// TIA Portal V19 export
TYPE "Tel393Out_PM"
// stored: Access Published
   STRUCT
      CU_STW1 : Struct   // Control word 1, Control Unit
         reserved_Bit08 : Bool;   // Reserved
         reserved_Bit09 : Bool;   // Reserved
         ackAutoSuppressed : Bool;   // Acknowledgment automatically suppressed
         reserved_Bit11 : Bool;   // Reserved
         masterSignOfLifeBit0 : Bool;   // Master sign-of-life bit 0
         masterSignOfLifeBit1 : Bool;   // Master sign-of-life bit 1
         masterSignOfLifeBit2 : Bool;   // Master sign-of-life bit 2
         masterSignOfLifeBit3 : Bool;   // Master sign-of-life bit 3
         syncFlag : Bool;   // This signal is used to synchonize the joint system time between the controller and drive unit BI: p 0681[0]
         rtcPing : Bool;   // This signal is used to set the UTC time using the Ping event BI: p 3104
         esrTrigger : Bool;   // ESR-Trigger
         reserved_Bit03 : Bool;   // Reserved
         reserved_Bit04 : Bool;   // Reserved
         reserved_Bit05 : Bool;   // Reserved
         reserved_Bit06 : Bool;   // Reserved
         acknowledge : Bool;   // 0 --> 1 = Acknowledge faults (Acknowledge fault. If the ON command is still active, the inverter switches to "closing lockout" state) p 2103[0] = r 2090.7
      END_STRUCT;
      A_DIGITAL : Struct   // Digital output (16-bit)
         reserved_Bit08 : Bool;   // Reserved
         reserved_Bit09 : Bool;   // Reserved
         reserved_Bit10 : Bool;   // Reserved
         reserved_Bit11 : Bool;   // Reserved
         reserved_Bit12 : Bool;   // Reserved
         reserved_Bit13 : Bool;   // Reserved
         reserved_Bit14 : Bool;   // Reserved
         reserved_Bit15 : Bool;   // Reserved
         digitalOutput8 : Bool;   // Digital output 8 (DI/DO 8); p0738 = r2091.0
         digitalOutput9 : Bool;   // Digital output 9 (DI/DO 9); p0739 = r2091.1
         digitalOutput10 : Bool;   // Digital output 10 (DI/DO 10); p0740 = r2091.2
         digitalOutput11 : Bool;   // Digital output 11 (DI/DO 11); p0741 = r2091.3
         digitalOutput12 : Bool;   // Digital output 12 (DI/DO 12); p0742 = r2091.4
         digitalOutput13 : Bool;   // Digital output 13 (DI/DO 13); p0743 = r2091.5
         digitalOutput14 : Bool;   // Digital output 14 (DI/DO 14); p0744 = r2091.6
         digitalOutput15 : Bool;   // Digital output 15 (DI/DO 15); p0745 = r2091.7
      END_STRUCT;
      A_DIGITAL_1 : Struct   // Digital output (16-bit)
         digitalOutput16 : Bool;   // Digital output 16 (DI/DO 16); p0746 = r2092.8
         reserved_Bit09 : Bool;   // Reserved
         reserved_Bit10 : Bool;   // Reserved
         reserved_Bit11 : Bool;   // Reserved
         reserved_Bit12 : Bool;   // Reserved
         reserved_Bit13 : Bool;   // Reserved
         reserved_Bit14 : Bool;   // Reserved
         reserved_Bit15 : Bool;   // Reserved
         "2ndacknowledge" : Bool;   // Set p2104 with r2092.0
         PathTestAxis1 : Bool;   // Set the Axis Stop test with r2092.1 from CU
         PathTestAxis2 : Bool;   // Set the Axis Stop test with r2092.2 from CU
         PathTestAxis3 : Bool;   // Set the Axis Stop test with r2092.3 from CU
         PathTestAxis4 : Bool;   // Set the Axis Stop test with r2092.4 from CU
         reserved_Bit05 : Bool;   // Reserved
         reserved_Bit06 : Bool;   // Reserved
         reserved_Bit07 : Bool;   // Reserved
      END_STRUCT;
      MT_STW : Struct   // Measuring probe control word
         risProbe1 : Bool;   // Activation of measuring time determination with the next rising edge
         risProbe2 : Bool;   // Activation of measuring time determination with the next rising edge
         risProbe3 : Bool;   // Activation of measuring time determination with the next rising edge
         risProbe4 : Bool;   // Activation of measuring time determination with the next rising edge
         risProbe5 : Bool;   // Activation of measuring time determination with the next rising edge
         risProbe6 : Bool;   // Activation of measuring time determination with the next rising edge
         risProbe7 : Bool;   // Activation of measuring time determination with the next rising edge
         risProbe8 : Bool;   // Activation of measuring time determination with the next rising edge
         falProbe1 : Bool;   // Activiation of measuring time determination with the next falling edge
         falProbe2 : Bool;   // Activiation of measuring time determination with the next falling edge
         falProbe3 : Bool;   // Activiation of measuring time determination with the next falling edge
         falProbe4 : Bool;   // Activiation of measuring time determination with the next falling edge
         falProbe5 : Bool;   // Activiation of measuring time determination with the next falling edge
         falProbe6 : Bool;   // Activiation of measuring time determination with the next falling edge
         falProbe7 : Bool;   // Activiation of measuring time determination with the next falling edge
         falProbe8 : Bool;   // Activiation of measuring time determination with the next falling edge
      END_STRUCT;
   END_STRUCT;
END_TYPE
